SUBAPPLICATION Button_Toggle_RPC_TO_Remote_BG_OPC (* IO-Diag-Taster (VT CButton) statt SoftKey: Loslassen (BT_RELEASED_UNLATCHED) ruft per CLIENT_0 einen argument- und rueckgabewertlosen OPC-UA-Methodenaufruf auf dem Zielmodul auf (reiner RPC-Trigger, kein AX_T_FF auf diesem Modul); GreenWhiteBackground zeigt den vom Zielmodul lokal ueberwachten Flipflop-Zustand. Identisches Protokoll wie Softkey_Toggle_RPC_TO_Remote_BG_OPC, nur Button_IE statt Softkey_IE (fuer Taster auf einer IO-Diag-DataMask statt einem SoftKey auf einer SoftKeyMask). *)
  (* Standard: 61499-2; Description: Copyright (c) 2026 Meisterschulen am Ostbahnhof This program and the accompanying materials are made available under the terms of the Eclipse Public License 2.0 which is available at https://www.eclipse.org/legal/epl-2.0/ SPDX-License-Identifier: EPL-2.0 *)
  (* Version 1.0, 2026-09-08, Franz Höpfinger, Meisterschulen am Ostbahnhof, initial API and implementation and/or initial documentation - Button-Analogon zu Softkey_Toggle_RPC_TO_Remote_BG_OPC, fuer IO-Diag-Taster (Q06/Q08 Freigabe-Toggle Aufnahme Links/Rechts) *)
  PACKAGE MyLib::sys;
  IMPORT isobus::UT::Q::const::IDs::ID_NULL;
  IMPORT isobus::UT::io::Button::ButtonActivationCode::BT_RELEASED_UNLATCHED;
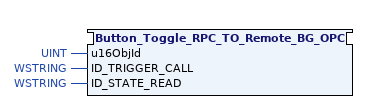
  VAR_INPUT
    u16ObjId : UINT := ID_NULL; (* Object ID Button/Background *)
    ID_TRIGGER_CALL : WSTRING; (* Remote-Methodenadresse (ACTION=CALL_METHOD) fuer den argumentlosen Trigger-Methodenaufruf auf dem Zielmodul *)
    ID_STATE_READ : WSTRING; (* Lokal ueberwachte Adresse (BOOL, ACTION=READ) fuer den Flipflop-Zustand, wird vom Zielmodul remote beschrieben *)
  END_VAR
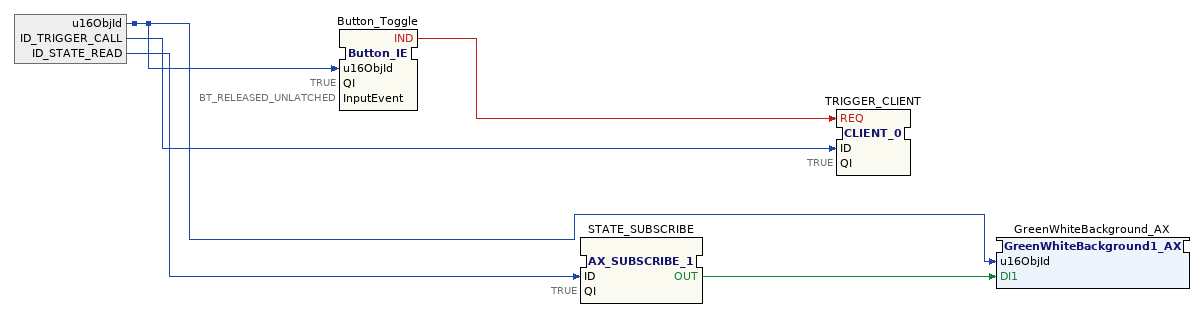
  FBS
    Button_Toggle : isobus::UT::io::Button::Button_IE(QI := TRUE, InputEvent := BT_RELEASED_UNLATCHED);
    TRIGGER_CLIENT : iec61499::net::CLIENT_0(QI := TRUE);
    STATE_SUBSCRIBE : adapter::net::AX_SUBSCRIBE_1(QI := TRUE);
  END_FBS
  SUBAPPS
    GreenWhiteBackground_AX : MyLib::sys::GreenWhiteBackground1_AX;
  END_SUBAPPS
  EVENT_CONNECTIONS
    Button_Toggle.IND TO TRIGGER_CLIENT.REQ;
  END_CONNECTIONS
  DATA_CONNECTIONS
    u16ObjId TO Button_Toggle.u16ObjId;
    u16ObjId TO GreenWhiteBackground_AX.u16ObjId;
    ID_TRIGGER_CALL TO TRIGGER_CLIENT.ID;
    ID_STATE_READ TO STATE_SUBSCRIBE.ID;
  END_CONNECTIONS
  ADAPTER_CONNECTIONS
    STATE_SUBSCRIBE.OUT TO GreenWhiteBackground_AX.DI1;
  END_CONNECTIONS
END_SUBAPPLICATION
